FUNCTION DisableSuctions : BOOL
VAR_IN_OUT
	suctionPads : ARRAY[*] OF SuctionPad;
END_VAR
VAR
	i : DINT;
END_VAR

FOR i:=LOWER_BOUND(suctionPads, 1) TO UPPER_BOUND(suctionPads, 1) BY 1 DO
	suctionPads[i].enable := FALSE;
END_FOR

END_FUNCTION

(* stored: Version 1.1.0.1, ProductVersion 3.1.4024.11
   POU DisableSuctions: Id {965b0722-98f5-4259-b855-fe92419145ac}, SpecialFunc None *)
